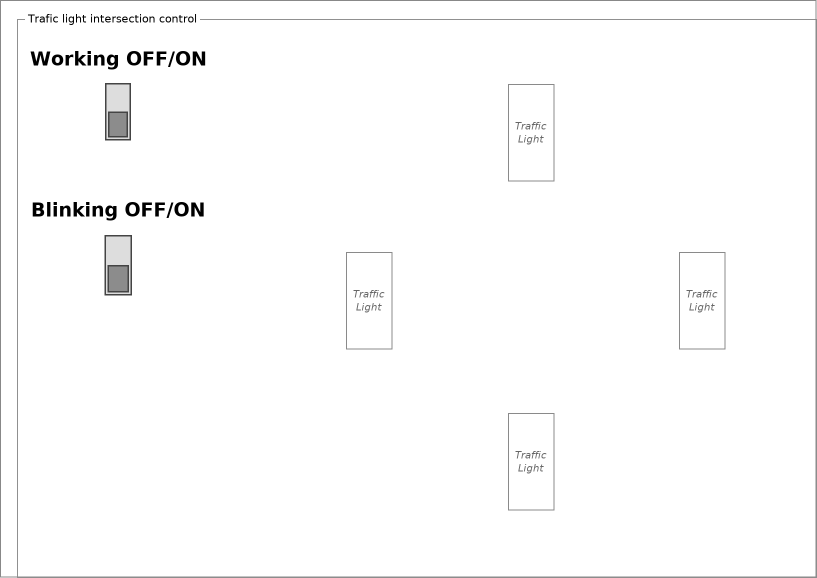
VISUALIZATION MainWindow  // 817x578
    GroupBox (17,11 800x567), "Trafic light intersection control"
        Rectangle (449,21 134x536), angle 90
        Label (14,33 175x30), "Working OFF/ON"
        Label (14,184 175x30), "Blinking OFF/ON"
        Line (395,120)
        Rectangle (449,19 134x536)
        Frame (491,73 46x97)
            shows TrafficLight(Red := MAIN.AutomationRunner.SignalControlledIntersectionAutomationUnit.TrafficLight2.RedLight.SimulatedContactValue, Yellow := MAIN.AutomationRunner.SignalControlledIntersectionAutomationUnit.TrafficLight2.YellowLight.SimulatedContactValue, Green := MAIN.AutomationRunner.SignalControlledIntersectionAutomationUnit.TrafficLight2.GreenLight.SimulatedContactValue)
        Frame (491,402 46x97)
            shows TrafficLight(Red := MAIN.AutomationRunner.SignalControlledIntersectionAutomationUnit.TrafficLight4.RedLight.SimulatedContactValue, Yellow := MAIN.AutomationRunner.SignalControlledIntersectionAutomationUnit.TrafficLight4.YellowLight.SimulatedContactValue, Green := MAIN.AutomationRunner.SignalControlledIntersectionAutomationUnit.TrafficLight4.GreenLight.SimulatedContactValue)
        Frame (662,241 46x97)
            shows TrafficLight(Red := MAIN.AutomationRunner.SignalControlledIntersectionAutomationUnit.TrafficLight3.RedLight.SimulatedContactValue, Yellow := MAIN.AutomationRunner.SignalControlledIntersectionAutomationUnit.TrafficLight3.YellowLight.SimulatedContactValue, Green := MAIN.AutomationRunner.SignalControlledIntersectionAutomationUnit.TrafficLight3.GreenLight.SimulatedContactValue)
        Frame (329,241 46x97)
            shows TrafficLight(Red := MAIN.AutomationRunner.SignalControlledIntersectionAutomationUnit.TrafficLight1.RedLight.SimulatedContactValue, Yellow := MAIN.AutomationRunner.SignalControlledIntersectionAutomationUnit.TrafficLight1.YellowLight.SimulatedContactValue, Green := MAIN.AutomationRunner.SignalControlledIntersectionAutomationUnit.TrafficLight1.GreenLight.SimulatedContactValue)
        DipSwitch (61,72 80x57), variable: MAIN.AutomationRunner.SignalControlledIntersectionAutomationUnit.WorkingModeSwitch.SimulatedContactValue, behaviour: TOGGLE, style: Switch-DipSwitch-Gray
        DipSwitch (61,224 80x60), variable: MAIN.AutomationRunner.SignalControlledIntersectionAutomationUnit.BlinkingYellowModeSwitch.SimulatedContactValue, behaviour: TOGGLE, style: Switch-DipSwitch-Gray
END_VISUALIZATION

(* stored: Version 1.1.0.1
   Visu MainWindow: Id {eac7b083-cabe-4cfa-a3a1-95d54c3932e1} *)
